TYPE ST_EL1809 :
STRUCT
	//--------------------------------------------------------------------------------------------------------
	sTerminalName                                           :   STRING(200):= 'EL1809 | 16-Channel Digital Input';
    //============================================================================================================================	
	// TERMINAL - EL1809 16-Channel Digital Input Terminal (Term 8)	
	iStartButoon                			AT %I*			: 	BOOL;	// EL1809 channel 1
	iStopButton                   			AT %I*			: 	BOOL;	// EL1809 channel 2
	iUP_OK        							AT %I*	 		: 	BOOL;	// EL1809 channel 3
	iUS_OK		   							AT %I*	 		: 	BOOL;	// EL1809 channel 4
	iPartPresentNest1         				AT %I*	 		: 	BOOL;	// EL1809 channel 5 		     			
	iPartPresentNest2 						AT %I*			: 	BOOL;	// EL1809 channel 6
	iPartPresentNest3               		AT %I*          :   BOOL;   // EL1809 channel 7 
    iPartPresentNest4          				AT %I*          :   BOOL;   // EL1809 channel 8
    iProcessCylinder1Retracted           	AT %I*          :   BOOL;   // EL1809 channel 9
	iProcessCylinder1Extended              	AT %I*          :   BOOL;   // EL1809 channel 10
	iProcessCylinder2Retracted              AT %I*          :   BOOL;   // EL1809 channel 11
	iProcessCylinder2Extended              	AT %I*          :   BOOL;   // EL1809 channel 12	   
	iRejectSensor         		   			AT %I*	 		: 	BOOL;	// EL1809 channel 13   
	iEL1809_Ch14       						AT %I*	 		: 	BOOL;	// EL1809 channel 14 
	iEL1809_Ch15							AT %I*			: 	BOOL;	// EL1809 channel 15  
	iEL1809_Ch16							AT %I*	 		: 	BOOL;	// EL1809 channel 16  	
	
	stTerminalInfo											: 	ST_Terminal_Info;

END_STRUCT
END_TYPE

(* stored: Version 1.1.0.1, ProductVersion 3.1.4024.13
   DUT ST_EL1809: Id {75a73e5d-4ca3-4f42-b76f-6978af3e18bb} *)
